FUNCTION_BLOCK FB_Vacuum
VAR_INPUT
	Vacuumsel:BYTE:=0;//0=真空和破真空都关，1=真空开，2=破真空开。
	tPTtime:TIME:=T#600MS;
END_VAR

VAR_IN_OUT
	VarrCyCtrl1			                  :ST_CyCtrl;//真空
	VarrCyCtrl2			                  :ST_CyCtrl;//破真空		
END_VAR

VAR
	ton:TON;	
END_VAR

ton(IN:= , PT:=tPTtime , Q=> , ET=> );
IF Vacuumsel=0  THEN
	VarrCyCtrl1.Cmd.bON:=VarrCyCtrl2.Cmd.bON:=FALSE;
	VarrCyCtrl1.Cmd.bOFF:=VarrCyCtrl2.Cmd.bOFF:=TRUE;
	ton.IN:=FALSE;
	Vacuumsel:=3;
ELSIF Vacuumsel=1 THEN
	VarrCyCtrl1.Cmd.bON:=VarrCyCtrl2.Cmd.bOFF:=TRUE;
	VarrCyCtrl1.Cmd.bOFF:=VarrCyCtrl2.Cmd.bON:=FALSE;
	ton.IN:=FALSE;
	Vacuumsel:=3;	
ELSIF Vacuumsel=2  THEN
	VarrCyCtrl1.Cmd.bON:=VarrCyCtrl2.Cmd.bOFF:=FALSE;
	VarrCyCtrl1.Cmd.bOFF:=VarrCyCtrl2.Cmd.bON:=TRUE;
	ton.IN:=TRUE;
	IF ton.Q THEN
		ton.IN:=FALSE;
		Vacuumsel:=0;
	END_IF	
END_IF

END_FUNCTION_BLOCK

(* stored: Version 1.1.0.1, ProductVersion 3.1.4024.12
   POU FB_Vacuum: Id {3a77ae25-5422-43c4-b585-e2abf0f96210}, SpecialFunc None *)
